Staubli VAL3: getLoaded.pgx

public program getLoaded(string& x_sLoaded[])
// get the loaded processList
begin
  // give back the actual saveCycle
  x_sLoaded=saveCycle:libPath()
  // empty the string if is the default
  if find(x_sLoaded,"template/saveCycle")!=-1
    x_sLoaded=""
  endIf
  // give back the program
  call getPath(x_sLoaded)
end
